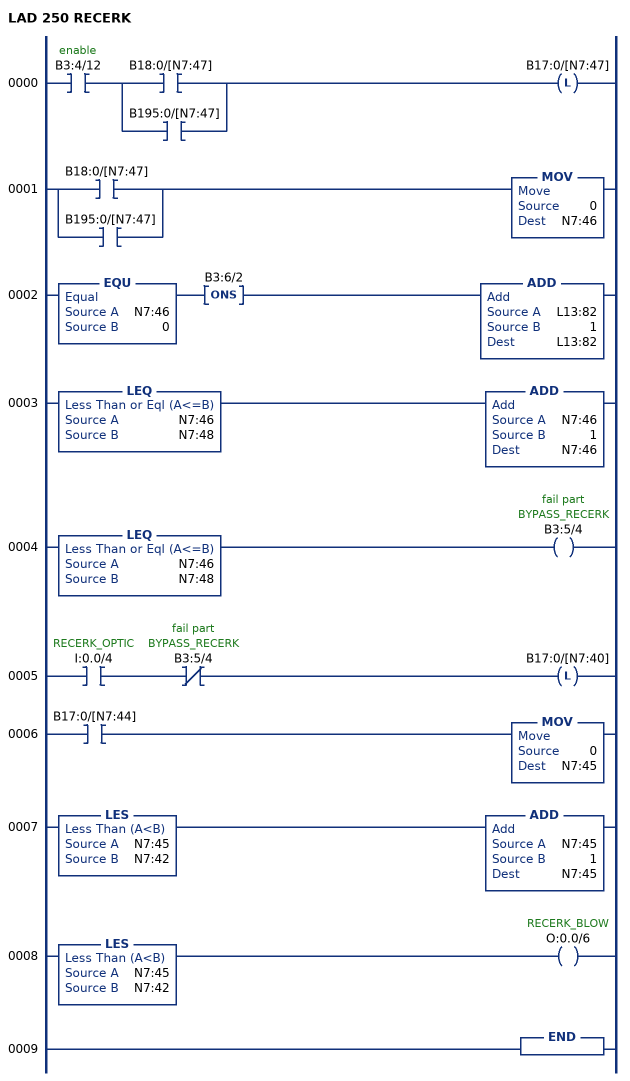
% Rung: 0 %
SOR XIC B3:4/12 BST XIC B18:0/[N7:47] NXB XIC B195:0/[N7:47] BND OTL B17:0/[N7:47] EOR
%   B3:4/12  "enable" %
%   B18:0  TOP_G %
%   N7:47  RECERK_BLOCKOPTIC_PT %
%   B195:0  TOP_NG %
%   B17:0  SIDE_G %
% Rung: 1 %
SOR BST XIC B18:0/[N7:47] NXB XIC B195:0/[N7:47] BND MOV 0 N7:46 EOR
%   B18:0  TOP_G %
%   N7:47  RECERK_BLOCKOPTIC_PT %
%   B195:0  TOP_NG %
% Rung: 2 %
SOR EQU N7:46 0 ONS B3:6/2 ADD L13:82 1 L13:82 EOR
% Rung: 3 %
SOR LEQ N7:46 N7:48 ADD N7:46 1 N7:46 EOR
%   N7:48  RECERK_BLK_BLOW_DIST %
% Rung: 4 %
SOR LEQ N7:46 N7:48 OTE B3:5/4 EOR
%   N7:48  RECERK_BLK_BLOW_DIST %
%   B3:5/4  BYPASS_RECERK  "fail part" %
% Rung: 5 %
SOR XIC I:0.0/4 XIO B3:5/4 OTL B17:0/[N7:40] EOR
%   I:0.0/4  RECERK_OPTIC %
%   B3:5/4  BYPASS_RECERK  "fail part" %
%   B17:0  SIDE_G %
%   N7:40  RECERK_OPTIC_POS %
% Rung: 6 %
SOR XIC B17:0/[N7:44] MOV 0 N7:45 EOR
%   B17:0  SIDE_G %
%   N7:44  RECERK_BLOW_POS  "adjusted for blow length" %
% Rung: 7 %
SOR LES N7:45 N7:42 ADD N7:45 1 N7:45 EOR
%   N7:42  RECERK_BLOW_LENGTH %
% Rung: 8 %
SOR LES N7:45 N7:42 OTE O:0.0/6 EOR
%   N7:42  RECERK_BLOW_LENGTH %
%   O:0.0/6  RECERK_BLOW %
% Rung: 9 %
SOR END EOR

LADDER 251 "RECERK SET"
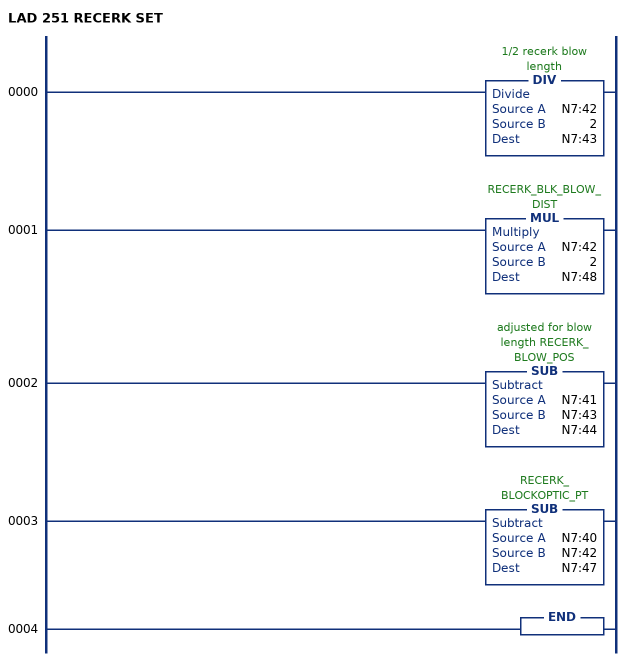
% Rung: 0 %
SOR DIV N7:42 2 N7:43 EOR
%   N7:42  RECERK_BLOW_LENGTH %
%   N7:43  "1/2 recerk blow length" %
% Rung: 1 %
SOR MUL N7:42 2 N7:48 EOR
%   N7:42  RECERK_BLOW_LENGTH %
%   N7:48  RECERK_BLK_BLOW_DIST %
% Rung: 2 %
SOR SUB N7:41 N7:43 N7:44 EOR
%   N7:41  RECERK_BLOW_POS_HMI  "recerk blow position set from hmi" %
%   N7:43  "1/2 recerk blow length" %
%   N7:44  RECERK_BLOW_POS  "adjusted for blow length" %
% Rung: 3 %
SOR SUB N7:40 N7:42 N7:47 EOR
%   N7:40  RECERK_OPTIC_POS %
%   N7:42  RECERK_BLOW_LENGTH %
%   N7:47  RECERK_BLOCKOPTIC_PT %
% Rung: 4 %
SOR END EOR

LADDER 252 "RATE1"
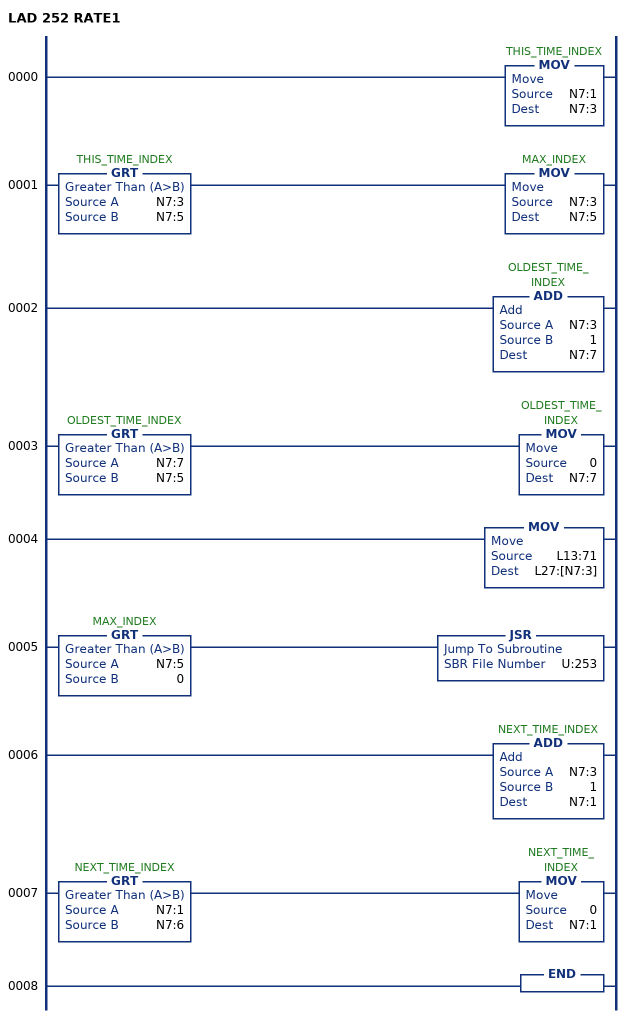
% Rung: 0 %
SOR MOV N7:1 N7:3 EOR
%   N7:1  NEXT_TIME_INDEX %
%   N7:3  THIS_TIME_INDEX %
% Rung: 1 %
SOR GRT N7:3 N7:5 MOV N7:3 N7:5 EOR
%   N7:3  THIS_TIME_INDEX %
%   N7:5  MAX_INDEX %
% Rung: 2 %
SOR ADD N7:3 1 N7:7 EOR
%   N7:3  THIS_TIME_INDEX %
%   N7:7  OLDEST_TIME_INDEX %
% Rung: 3 %
SOR GRT N7:7 N7:5 MOV 0 N7:7 EOR
%   N7:7  OLDEST_TIME_INDEX %
%   N7:5  MAX_INDEX %
% Rung: 4 %
SOR MOV L13:71 L27:[N7:3] EOR
%   L13:71  HSC_TIME %
%   N7:3  THIS_TIME_INDEX %
% Rung: 5 %
SOR GRT N7:5 0 JSR U:253 EOR
%   N7:5  MAX_INDEX %
% Rung: 6 %
SOR ADD N7:3 1 N7:1 EOR
%   N7:3  THIS_TIME_INDEX %
%   N7:1  NEXT_TIME_INDEX %
% Rung: 7 %
SOR GRT N7:1 N7:6 MOV 0 N7:1 EOR
%   N7:1  NEXT_TIME_INDEX %
%   N7:6  UPPER_INDEX_LIMIT  "buffer count 1" %
% Rung: 8 %
SOR END EOR

LADDER 253 "RATE2"
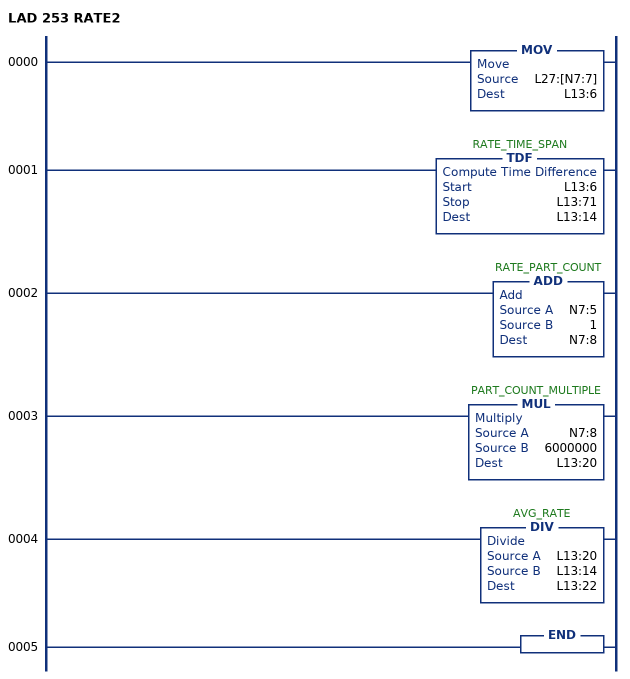
% Rung: 0 %
SOR MOV L27:[N7:7] L13:6 EOR
%   N7:7  OLDEST_TIME_INDEX %
% Rung: 1 %
SOR TDF L13:6 L13:71 L13:14 EOR
%   L13:71  HSC_TIME %
%   L13:14  RATE_TIME_SPAN %
% Rung: 2 %
SOR ADD N7:5 1 N7:8 EOR
%   N7:5  MAX_INDEX %
%   N7:8  RATE_PART_COUNT %
% Rung: 3 %
SOR MUL N7:8 6000000 L13:20 EOR
%   N7:8  RATE_PART_COUNT %
%   L13:20  PART_COUNT_MULTIPLE %
% Rung: 4 %
SOR DIV L13:20 L13:14 L13:22 EOR
%   L13:20  PART_COUNT_MULTIPLE %
%   L13:14  RATE_TIME_SPAN %
%   L13:22  AVG_RATE %
% Rung: 5 %
SOR END EOR

LADDER 254 "RESET RATE"
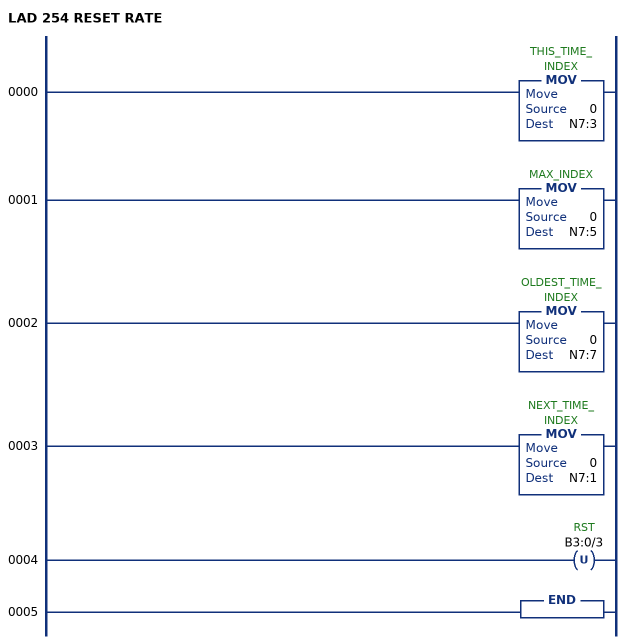
% Rung: 0 %
SOR MOV 0 N7:3 EOR
%   N7:3  THIS_TIME_INDEX %
% Rung: 1 %
SOR MOV 0 N7:5 EOR
%   N7:5  MAX_INDEX %
% Rung: 2 %
SOR MOV 0 N7:7 EOR
%   N7:7  OLDEST_TIME_INDEX %
% Rung: 3 %
SOR MOV 0 N7:1 EOR
%   N7:1  NEXT_TIME_INDEX %
% Rung: 4 %
SOR OTU B3:0/3 EOR
%   B3:0/3  RST %
% Rung: 5 %
SOR END EOR

LADDER 255 "UNUSED"
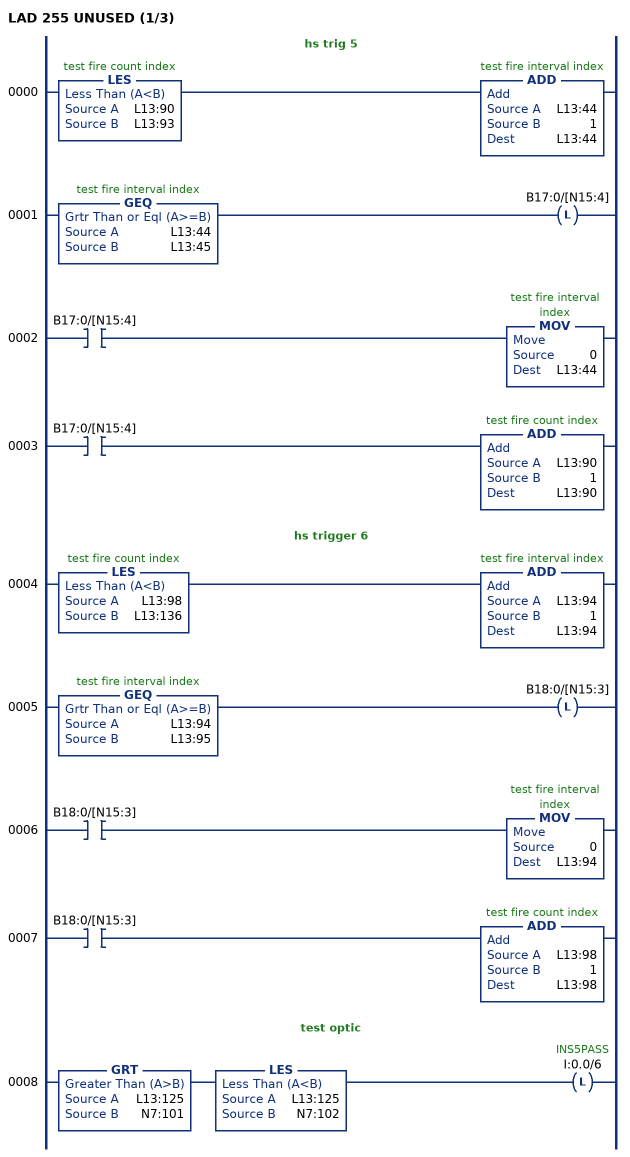
% Rung: 0 %
% TITLE: hs trig 5 %
SOR LES L13:90 L13:93 ADD L13:44 1 L13:44 EOR
%   L13:90  "test fire count index" %
%   L13:93  "test fire count" %
%   L13:44  "test fire interval index" %
% Rung: 1 %
SOR GEQ L13:44 L13:45 OTL B17:0/[N15:4] EOR
%   L13:44  "test fire interval index" %
%   L13:45  "test fire interval" %
%   B17:0  SIDE_G %
%   N15:4  INS_5_TRIG_LOC %
% Rung: 2 %
SOR XIC B17:0/[N15:4] MOV 0 L13:44 EOR
%   B17:0  SIDE_G %
%   N15:4  INS_5_TRIG_LOC %
%   L13:44  "test fire interval index" %
% Rung: 3 %
SOR XIC B17:0/[N15:4] ADD L13:90 1 L13:90 EOR
%   B17:0  SIDE_G %
%   N15:4  INS_5_TRIG_LOC %
%   L13:90  "test fire count index" %
% Rung: 4 %
% TITLE: hs trigger 6 %
SOR LES L13:98 L13:136 ADD L13:94 1 L13:94 EOR
%   L13:98  "test fire count index" %
%   L13:136  "test fire count" %
%   L13:94  "test fire interval index" %
% Rung: 5 %
SOR GEQ L13:94 L13:95 OTL B18:0/[N15:3] EOR
%   L13:94  "test fire interval index" %
%   L13:95  "test fire interval" %
%   B18:0  TOP_G %
%   N15:3  INS_6_TRIG_LOC %
% Rung: 6 %
SOR XIC B18:0/[N15:3] MOV 0 L13:94 EOR
%   B18:0  TOP_G %
%   N15:3  INS_6_TRIG_LOC %
%   L13:94  "test fire interval index" %
% Rung: 7 %
SOR XIC B18:0/[N15:3] ADD L13:98 1 L13:98 EOR
%   B18:0  TOP_G %
%   N15:3  INS_6_TRIG_LOC %
%   L13:98  "test fire count index" %
% Rung: 8 %
% TITLE: test optic %
SOR GRT L13:125 N7:101 LES L13:125 N7:102 OTL I:0.0/6 EOR
%   I:0.0/6  INS5PASS %

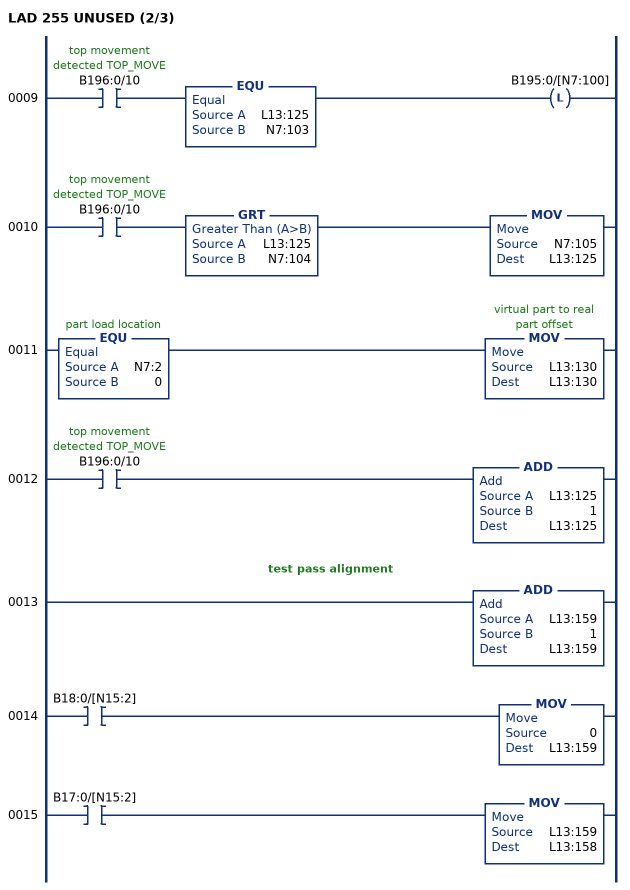
% Rung: 9 %
SOR XIC B196:0/10 EQU L13:125 N7:103 OTL B195:0/[N7:100] EOR
%   B196:0/10  TOP_MOVE  "top movement detected" %
%   B195:0  TOP_NG %
% Rung: 10 %
SOR XIC B196:0/10 GRT L13:125 N7:104 MOV N7:105 L13:125 EOR
%   B196:0/10  TOP_MOVE  "top movement detected" %
% Rung: 11 %
SOR EQU N7:2 0 MOV L13:130 L13:130 EOR
%   N7:2  "part load location" %
%   L13:130  "virtual part to real part offset" %
% Rung: 12 %
SOR XIC B196:0/10 ADD L13:125 1 L13:125 EOR
%   B196:0/10  TOP_MOVE  "top movement detected" %
% Rung: 13 %
% TITLE: test pass alignment %
SOR ADD L13:159 1 L13:159 EOR
% Rung: 14 %
SOR XIC B18:0/[N15:2] MOV 0 L13:159 EOR
%   B18:0  TOP_G %
%   N15:2  BLOW_PT %
% Rung: 15 %
SOR XIC B17:0/[N15:2] MOV L13:159 L13:158 EOR
%   B17:0  SIDE_G %
%   N15:2  BLOW_PT %

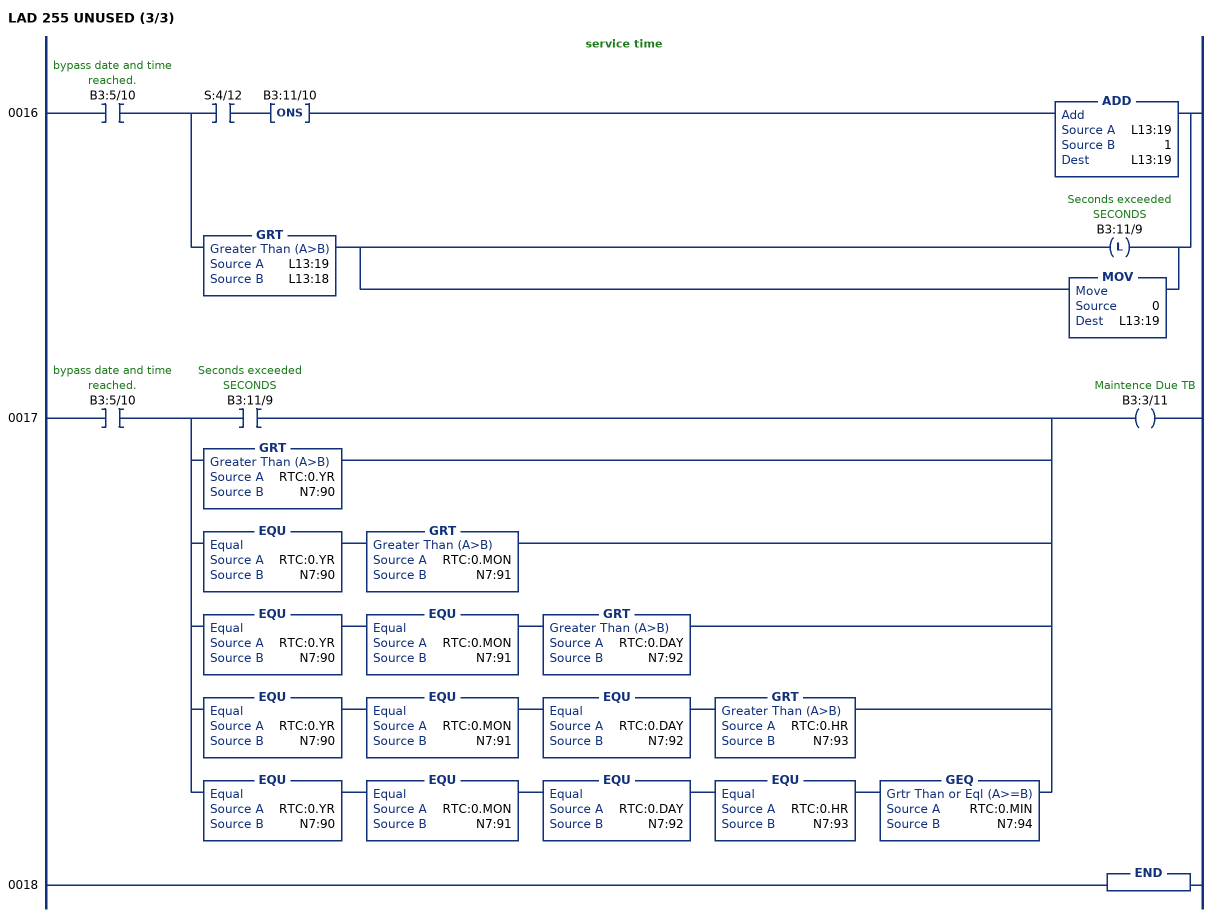
% Rung: 16 %
% TITLE: service time %
SOR XIC B3:5/10 BST XIC S:4/12 ONS B3:11/10 ADD L13:19 1 L13:19 NXB GRT L13:19 L13:18 BST OTL B3:11/9 NXB MOV 0 L13:19 BND BND EOR
%   B3:5/10  "bypass date and time reached." %
%   L13:18  MAX %
%   B3:11/9  SECONDS  "Seconds exceeded" %
% Rung: 17 %
SOR XIC B3:5/10 BST XIC B3:11/9 NXB GRT RTC:0.YR N7:90 NXB EQU RTC:0.YR N7:90 GRT RTC:0.MON N7:91 NXB EQU RTC:0.YR N7:90 EQU RTC:0.MON N7:91 GRT RTC:0.DAY N7:92 NXB EQU RTC:0.YR N7:90 EQU RTC:0.MON N7:91 EQU RTC:0.DAY N7:92 GRT RTC:0.HR N7:93 NXB EQU RTC:0.YR N7:90 EQU RTC:0.MON N7:91 EQU RTC:0.DAY N7:92 EQU RTC:0.HR N7:93 GEQ RTC:0.MIN N7:94 BND OTE B3:3/11 EOR
%   B3:5/10  "bypass date and time reached." %
%   B3:11/9  SECONDS  "Seconds exceeded" %
%   N7:90  RTC %
%   B3:3/11  TB  "Maintence Due" %
% Rung: 18 %
SOR END EOR

OTHER DOCUMENTED ADDRESSES
  B12:0/1  FELL_PARTS_FAULT
  B196:1/2  DOWNTRACK_OPTIC_RUN  "Feed Bowl optic Run Signal after timing delays"
  I:0.0/0  TOP_CONV_ENC_A
  I:0.0/1  TOP_CONV_ENC_B
  I:0.7  "Air Presure Sensor Input Signal"
  L13:61  "max acquisition time in ms"
  L42:0/2  "box full read (unused)"
  L42:1/1  "ps stop write (unused)"
  L183:3  L  "button state"
  N7:35  "maximum buffers"
  N15:9  FEED_WHEEL_STOP_TIME
  N197:7  "down track on delay"
  N197:8  "down track off delay"
  O:0.0/0  "spare"
  O:0.0/1  "spare"
  O:0.0/10  "spare"
  O:0.0/11  "spare"
  PFILE:6  "check for part jams"
  PFILE:10  "Bottom belt HSC"
  PFILE:12  "Top belt HSC"
  Q2:55  END_OF_MAIN
  T4:6  FEED_WHEEL_OFF_TIMER  "Delay to shut off feed wheel"
  U:6  "feed"
  U:217  "test trigger"

COMMENTS NOT ATTACHED TO A CURRENT RUNG
  F8:13: *************************
    Loads Side Camera Passing data into a bit shift
    *************************
    
    loads passing data bit into passing data bit shift register at the part present cl.
  I:0.0/8: special rung for testing. This rung can simulate a pass signal. It will not be timed correctly.
  B23:0/0: Yet another bit shift load with data in the part position indicating that there was a bottom system part pass as well as a top system part present at this location.
    
    verified works w/bypassed 071910 and unbypassed 072010
  C5:4: tempory counting to verify pass part count with boxing part count.
  B22:0/0: ***********************
     Bottom Part Syncronizing Logic
    ***********************
    
    This is the point at the bottom of the top conveyor where the part jumps from the bottom conveyor.  This system will then track the part through the top system to the point of the laser optic in order to verify that the part in question has passed the bottom inspection.  I believe that we NEED to include FAILING inspections to eliminate the possibility of a out of position part from passing. LW 072010
  T20:2.ACC: This rung is starting a timer that should be activated directly before the laser optic part presense sensor on the top conveyer and should cause the top optic to be ignored if the bottom camera system didn't pass. however other arrangements must be made if the bottom camera isn't going to be used as is the case with a nut inspection.
  T20:2: The timer used to verify that the part that triggered the top laser optic has passed the bottom camer. needs to be count
  N17:8: ****************************************************************************************************************
    I can not find anywhere in the program where the "Test Spacing From Pickup to Trigger is activated indicating to me that this entire function must not be doing anything in this program at this time.
    ****************************************************************************************************************
  B11:0/0: load part present bit shit with one shot data from the part present sensor
  B3:7/9: ************************************
     The next 3 rungs appear to do nothing
    ***********************************
  B3:6/1: ***********************
    Part Width and  Location
    ***********************
    
    Calculates the position of parts on the top belt by measureing the part width by calculating the number of belt movement pulses that occure when the optic is blocked and then devides that in half and add that to the optic location in the part presnet bit shift when the top optic is cleared.
  B9:0/[N7:47]: Remove any part present signals outside of expected location
  B9:0/[N7:50]: Remove any part present signals outside of expected location
  F19:0: Counter inside of a high speed counter interrupt counts the number of Bit Shifts that need to be processed in order to move the logic with the parts on the conveyor.
  F8:14: **************
    Bottom Top Camera Trigger
    *************
    
    Trigger Bottom Top Camera
  N10:4: test if boxing is connected
  B3:11/3: After initial delay allow blow two start functioning
  RUNG000150-000011: trigger count
  RUNG000150-000012: wipe stored part data if acq time expires
  RUNG000150-000013: clear data for aquire time expired
  RUNG000150-000014: clear data for time
  RUNG000150-000016: wiped count
  RUNG000150-000018: pass, fail and acquire inputs
  RUNG000150-000025: pass code / Set pass bit in Bit Shift
    captures result position and processing time
    Unlatch pass bit
  RUNG000150-000032: pass count
  RUNG000150-000035: fail count
  RUNG000150-000038: acquire code
  RUNG000150-000039: Grab trigger/acquire position
    Grab acquire time
  RUNG000150-000041: transfer tracked part positon from trigger/acquire to the acquire/result
    capture acquire time
    reset process time
  L14:8: on when ok for run
  L14:3: off when ok to run
  L14:2: off when ok to run
  L14:5: on when ok to run, rear off turns both off
  L13:165: maximum q i1
  N7:76: removed relieance on trigger signal
  N197:20/0: Passes deformed head blowoff command to TOP PLC where solenoid output is located.
  L13:162: maximum q
  L13:163: maximum average q
  B3:10/1: prevents momentary signals from box present sensor from tripping the logic for box not present
    
    This is in responce to a problem created by the sensor occasionally turning on as if no box was in its path when there is a box present.
  B3:6/2: IF PROCESSING FAULT OCURES AT COUNTER SENSOR; CLEAR THE BELT OF PASSING DATA
  L14:23: ****************  nEEDS fIXING  **********************
  L14:36: ****************  nEEDS fIXING  **********************
  RUNG000010-000014: ****
                      Zeros out the non passing part count when one passes
    ****
  RUNG000010-000018: Remove any part present signals outside of expected location
  T4:27: Check for buffer reset
  T4:26: Check for buffer reset
  RUNG000125-000014: clear data for time
  RUNG000125-000013: clear data for aquire time expired
  RUNG000125-000012: wipe stored part data if acq time expires
  RUNG000125-000011: trigger count
  RUNG000125-000029: Set pass bit in Bit Shift
    captures result position and processing time
    Unlatch pass bit
  RUNG000125-000027: transfer tracked part positon from trigger/acquire to the acquire/result
    capture acquire time
    reset process time
  RUNG000125-000026: Grab trigger/acquire position
    Grab acquire time
  RUNG000125-000025: pass code / Set pass bit in Bit Shift
    captures result position and processing time
    Unlatch pass bit
  RUNG000125-000018: pass, fail and acquire inputs
  RUNG000125-000016: wiped count

REVISION NOTES
  13: updated count reset
  14: added io moduals
  15: multiple steps toward new hmi integration
  21: test

DATA TABLE (non-zero values as saved)
DATA B3
% B3:0 % 0XA001 0X5060 0X02C4 0XA008 0X8B26 0X0341 0XA881 0X659A 0X4130 0X0000
% B3:10 % 0X2041 0X0846 0X2000 0X0000 0X0000 0X0000 0X0000 0X0000 0X0000 0X0000
DATA T4
% .PRE .ACC %
% T4:0 % 333 163
% T4:1 % 333 290
% T4:2 % 600 0
% T4:3 % 1000 1002
% T4:4 % 3 1
% T4:5 % 666 0
% T4:6 % 10 32766
% T4:7 % 250 0
% T4:8 % 250 0
% T4:9 % 50 3
% T4:10 % 200 0
% T4:11 % 666 0
% T4:12 % 14 29
% T4:13 % 6 4
% T4:14 % 250 0
% T4:15 % 333 30
% T4:16 % 333 19
% T4:17 % 100 64
% T4:18 % 120 120
% T4:19 % 300 0
% T4:20 % 200 0
% T4:21 % 200 0
% T4:22 % 200 0
% T4:23 % 250 0
% T4:24 % 666 0
% T4:25 % 666 0
% T4:26 % 250 0
% T4:27 % 250 0
% T4:28 % 250 0
% T4:29 % 5000 0
% T4:30 % 50 50
% T4:31 % 20 0
% T4:32 % 69 0
DATA C5
% .PRE .ACC %
% C5:0 % 32766 0
DATA R6
% .LEN .POS %
% R6:0 % 2048 0
% R6:1 % 2048 0
% R6:2 % 3 0
% R6:3 % 3 0
% R6:4 % 1250 0
% R6:5 % 1250 0
% R6:6 % 1300 0
% R6:7 % 10 0
% R6:8 % 3 0
% R6:9 % 3 0
% R6:10 % 1440 0
% R6:11 % 1440 0
% R6:12 % 10 0
% R6:13 % 10 0
% R6:14 % 10 0
% R6:15 % 10 0
% R6:16 % 1300 0
% R6:17 % 1440 0
% R6:18 % 1440 0
% R6:19 % 10 0
DATA N7
% N7:0 % 11069 27 1164 26 0 26 49 0 27 0
% N7:10 % 40 70 0 40 1512 250 777 666 10632 94
% N7:20 % 9591 93 9543 0 0 12 12 1580 333 20
% N7:30 % 46 10 2 20 46 10 1503 333 1493 333
% N7:40 % 2067 2122 40 20 2102 40 81 2027 80 1515
% N7:50 % 1520 400 27 14 0 0 32767 1520 28 15
% N7:60 % 1 1 4012 20 31 0 0 15 30 20
% N7:70 % 0 21 23 27738 32767 0 122 0 16 0
% N7:80 % 0 6 95 0 0 0 5 500 0 0
% N7:90 % 2011 4 4 12 1 0 0 0 0 1600
% N7:100 % 1003 90 110 100 175 25 0 0 0 0
DATA F8
% F8:0 % 18 206.64 23807 499 0.23807
% F8:5 % 0 0 500 1.9 2
% F8:10 % 1 0.08897486 0 101 63.26563
% F8:15 % 37.73437 4040 2 0 0
% F8:20 % 0 0.02 0 1 0
% F8:25 % 0 932781 0.222 279.6551 848597
% F8:30 % 0 170 0.03 38 852060
% F8:35 % 0 0 0 0 77
% F8:40 % 101 37.73437 0 100 1
% F8:45 % 1 2 0.21455 0 0
% F8:50 % 0 0 1 0 1
% F8:55 % 2000000 -221 0 0 0
% F8:95 % 0 0 0 492 4.92
DATA B12
% B12:0 % 0X0454 0X0000 0X0000 0X0000 0X0000 0X0000 0X0000 0X0000 0X0000 0X0000
DATA L13
% L13:0 % 308402300 308407124 4824 0 1000
% L13:5 % 1 -75983992 100 1162124017 1162124017
% L13:10 % 492 21600 28709 0 1030982652
% L13:15 % 350704886 -2147483648 2147483647 2147483647 82058
% L13:20 % 162000000 1592451203 0 320903532 1592451203
% L13:25 % 319 0 29801374 5 1000000000
% L13:30 % -344351 28623 1591069087 84 57344
% L13:35 % 0 57344 1591069087 1 1592451203
% L13:40 % -366691798 0 8 20 0
% L13:45 % 60 700 1 0 33
% L13:50 % 0 20 444 20 444
% L13:55 % 0 585 18048 10764 336
% L13:60 % 0 3300 84 2147483647 0
% L13:65 % 0 20 0 1926950760 1
% L13:70 % 955102215 955102183 32 0 2400
% L13:75 % -2 0 1072712 320903515 1073
% L13:80 % 319 -94 5615 0 2
% L13:85 % 6475 180 17292 344402 -463410
% L13:90 % 26616 0 0 1000 0
% L13:95 % 60 336 674 25989 350360221
% L13:100 % 351168041 -464527 -5036228 342295039 216
% L13:105 % 1592278120 1592278120 173083 0 537010368
% L13:110 % 6 1195 556 1590168231 1592376160
% L13:115 % 1592376187 27 14 1592376173 2207942
% L13:120 % 1195 3421 0 30 556
% L13:125 % 164 1592278120 1592278120 20 46
% L13:130 % 2207942 31204 31135 336 0
% L13:135 % 0 1000 337 12 0
% L13:140 % 12 6391320 12 0 20
% L13:145 % 64 1273 1284 111 111
% L13:150 % -1538760531 -1538760111 88 0 100
% L13:155 % 420 332 24 0 168160
% L13:160 % 3 18 4 395082 53203921
% L13:165 % 3 189116 95 13 8150
% L13:170 % 55946610 30 2868678 342419 0
% L13:175 % 0 0 45 32 38
% L13:180 % 176247033 25 99000 52866 644409
% L13:185 % 64 916459 92 627156 63
% L13:190 % 4 5 0 0 0
DATA F14
% F14:0 % 760.1599 200.1099 76 20 15
% F14:5 % 32766 21297.9 0 0 0
DATA N15
% N15:0 % 6 889 1976 1512 1502 134 100 1172 1150 10
% N15:10 % 61 504 0 0 0 0 1172 0 0 0
DATA L16
% L16:0 % 8 14 11 0 20
% L16:5 % 250 5000 5000 182 19
% L16:10 % 1256 18 2045 6599584 98
% L16:15 % 99 0 0 0 0
DATA B17
% B17:60 % 0XC000 0X0000 0X0000 0X0000 0X0000 0X0000 0X0000 0X0000 0X0000 0X0000
DATA B18
% B18:60 % 0XC000 0X0000 0X0000 0X0000 0X0000 0X0000 0X0000 0X0000 0X0000 0X0000
DATA L19
% L19:0 % -469940 -468592 -468256 -466907 -466571
% L19:5 % -465222 -464883 -381237 -380973 -380903
% L19:10 % -380854 -355115 -344351 -500587 -500251
% L19:15 % -498902 -498565 -497218 -496882 -495534
% L19:20 % -495198 -493853 -493515 -492169 -491833
% L19:25 % -490486 -490150 -488802 -488465 -487117
% L19:30 % -486780 -485430 -485093 -483747 -483408
% L19:35 % -482062 -481724 -480377 -480039 -478693
% L19:40 % -478357 -477010 -476673 -475325 -474988
% L19:45 % -473642 -473303 -471957 -471622 -470277
DATA L20
% L20:0 % 1592278120 1592278120 1592278120 1592278120 1592278120
% L20:5 % 1592278120 1592278120 1592294886 1592294950 1592294967
% L20:10 % 1592294979 1592301197 1592303799 1592278120 1592278120
% L20:15 % 1592278120 1592278120 1592278120 1592278120 1592278120
% L20:20 % 1592278120 1592278120 1592278120 1592278120 1592278120
% L20:25 % 1592278120 1592278120 1592278120 1592278120 1592278120
% L20:30 % 1592278120 1592278120 1592278120 1592278120 1592278120
% L20:35 % 1592278120 1592278120 1592278120 1592278120 1592278120
% L20:40 % 1592278120 1592278120 1592278120 1592278120 1592278120
% L20:45 % 1592278120 1592278120 1592278120 1592278120 1592278120
DATA L21
% L21:0 % 242620121 242621467 242621803 242623146 242623482
% L21:5 % 242624823 242625160 242626503 242626839 242628182
% L21:10 % 242628517 242629860 242630195 242631539 242631874
% L21:15 % 242633220 242633556 242634900 242635236 242636581
% L21:20 % 242636916 242638260 242638595 242822056 242822392
% L21:25 % 242822728 242823065 242823400 242823737 242824074
% L21:30 % 257003035 257003370 257003706 257005050 320901516
% L21:35 % 320901853 320902189 320902525 320902860 320903196
% L21:40 % 320903532 242613067 242613403 242614746 242615083
% L21:45 % 242616426 242616761 242618104 242618440 242619785
DATA L22
% L22:0 % 1592451203 1592451203 1592451203 1592451203 1592451203
% L22:5 % 1592451203 1592451203 1592451203 1592451203 1592451203
% L22:10 % 1592451203 1592451203 1592451203 1592451203 1592451203
% L22:15 % 1592451203 1592451203 1592451203 1592451203 1592451203
% L22:20 % 1592451203 1592451203 1592451203 1592451203 1592451203
% L22:25 % 1592451203 1592451203 1592451203 1592451203 1592451203
% L22:30 % 1592451203 1592451203 1592451203 1592451203 1592451203
% L22:35 % 1592451203 1592451203 1592451203 1592451203 1592451203
% L22:40 % 1592451203 1592451203 1592451203 1592451203 1592451203
% L22:45 % 1592451203 1592451203 1592451203 1592451203 1592451203
DATA L23
% L23:0 % 321208 322551 322887 324232 324567
% L23:5 % 325913 326249 327593 327929 329273
% L23:10 % 329610 330955 331291 332634 332970
% L23:15 % 334315 334651 335996 336332 337677
% L23:20 % 338014 339359 339694 341041 341377
% L23:25 % 342721 343058 344402 344738 304058
% L23:30 % 304394 305741 306077 307423 307759
% L23:35 % 309105 309442 310787 311123 312467
% L23:40 % 312803 314147 314482 315827 316163
% L23:45 % 317508 317844 319190 319527 320871
DATA L24
% L24:0 % 1592447007 1592447007 1592447007 1592447007 1592447007
% L24:5 % 1592447007 1592447007 1592447007 1592447007 1592447007
% L24:10 % 1592447007 1592447007 1592447007 1592447007 1592447007
% L24:15 % 1592447007 1592447007 1592447007 1592447007 1592447007
% L24:20 % 1592447007 1592447007 1592447007 1592447007 1592447007
% L24:25 % 1592447007 1592447007 1592447007 1592447007 1592447007
% L24:30 % 1592447007 1592447007 1592447007 1592447007 1592447007
% L24:35 % 1592447007 1592447007 1592447007 1592447007 1592447007
% L24:40 % 1592447007 1592447007 1592447007 1592447007 1592447007
% L24:45 % 1592447007 1592447007 1592447007 1592447007 1592447007
DATA L25
% L25:0 % -475206 -474868 -473520 -473183 -471837
% L25:5 % -471500 -470152 -469816 -468467 -468130
% L25:10 % -466782 -466444 -465096 -464759 -463410
% L25:15 % -463073 -503828 -503490 -502145 -501808
% L25:20 % -500462 -500127 -498781 -498444 -497099
% L25:25 % -496762 -495417 -495082 -493735 -493398
% L25:30 % -492050 -491712 -490368 -490032 -488687
% L25:35 % -488351 -487003 -486667 -485317 -484980
% L25:40 % -483630 -483292 -481947 -481608 -480262
% L25:45 % -479926 -478576 -478238 -476890 -476553
DATA L26
% L26:0 % 1592278120 1592278120 1592278120 1592278120 1592278120
% L26:5 % 1592278120 1592278120 1592278120 1592278120 1592278120
% L26:10 % 1592278120 1592278120 1592278120 1592278120 1592278120
% L26:15 % 1592278120 1592278120 1592278120 1592278120 1592278120
% L26:20 % 1592278120 1592278120 1592278120 1592278120 1592278120
% L26:25 % 1592278120 1592278120 1592278120 1592278120 1592278120
% L26:30 % 1592278120 1592278120 1592278120 1592278120 1592278120
% L26:35 % 1592278120 1592278120 1592278120 1592278120 1592278120
% L26:40 % 1592278120 1592278120 1592278120 1592278120 1592278120
% L26:45 % 1592278120 1592278120 1592278120 1592278120 1592278120
DATA L27
% L27:0 % -75983992 -75957196 -75956598 -75951544 -75950734
% L27:5 % -75947930 -75946415 -75945812 -75944870 -75943992
% L27:10 % -75941967 -75939459 -75934924 -75898731 -75897730
% L27:15 % -73346188 -72261338 -72201767 -68929091 -59219708
% L27:20 % -55819289 -53892544 -50990397 -48812047 -45021425
% L27:25 % -43383575 -41958136 502552452 531598359 531633864
% L27:30 % 531668449 531704205 531755229 531795341 531997256
% L27:35 % 625725685 625797461 627329145 627380790 627425916
% L27:40 % 627475622 627507784 627530557 627557972 627592344
% L27:45 % 627654448 627674800 627694163 627713711 627733603
DATA L42
% L42:0 % 8 256 0 0 0
% L42:5 % 45 45 45 0 0
% L42:20 % 0 0 32766 32766 0
% L42:50 % 0 30
DATA L183
% L183:0 % 1427522383 1427522384 1 1000000000 0
% L183:5 % 321 6 283 0 0
DATA N184
% N184:0 % 0 333 0 0 0 0 0 0 0 0
DATA B185
% B185:0 % 0X0200 0X0001 0X0000 0X0000 0X0000 0X0000 0X0000 0X0000 0X0000 0X0000
DATA N186
% N186:0 % 100 0 0 0 0 0 0 0 0 0
DATA L187
% L187:0 % 34 0 497 0 0
% L187:5 % 1063 0 0 0 0
DATA F188
% F188:0 % 6 66 11 44 29
DATA B189
% B189:0 % 0X00F0 0X0000 0X0000 0X0000 0X0000 0X0000 0X0000 0X0000 0X0000 0X0000
DATA L190
% L190:0 % 1 5 0 0 0
% L190:30 % 0 2 0 0 0
DATA B191
% B191:0 % 0X0000 0X0001 0X0000 0X0000 0X0000 0X0000 0X0000 0X0000 0X0000 0X0000
DATA L192
% L192:0 % -1444152502 266932201 5055 76 0
% L192:5 % 1000000 39200000 999 999 8
% L192:10 % 0 0 0 78 17
% L192:15 % 1926950760 332250347 860888 0 0
% L192:20 % 180 0 0 0 0
DATA F193
% F193:0 % 1.268652 0.315 0.022 6 760
% F193:5 % -0.8252563 0.2 -0.1650513 964.1756 31592.18
% F193:10 % 0.011 0.195 0.165 0.337 200
% F193:15 % 0.09407043 0.025 0.002351761 0 1092.66
DATA B196
% B196:0 % 0X0224 0X9FF2 0X0001 0X0000 0X0000 0X0000 0X0000 0X0000 0X0000 0X0000
% B196:30 % 0XE800 0X9BFF 0XEBFF 0XFFDF 0XFFFF 0X0000 0X0000 0X0000 0X0000 0X0000
DATA N197
% N197:0 % 1560 150 500 2500 2500 14417 5555 300 150 0
% N197:10 % 4000 969 4 0 0 0 0 0 0 0
% N197:30 % 15 48 0 0 0 0 0 0 0 0
DATA B198
% B198:0 % 0X0009 0X0000 0X0000 0X0000 0X0000 0X0000 0X0000 0X0000 0X0000 0X0000
DATA L199
% L199:0 % 1 5571998 134 11 3579521
% L199:5 % 0 0 0 5 43136
% L199:10 % 0 224 10256 556 0
% L199:15 % 0 0 0 278717848 518
% L199:20 % 28295 16430853 5001 5001 0
% L199:25 % 0 0 28329 1 3781224
% L199:30 % 21630086 251 3809367 15030467 111
% L199:35 % 555 555 0 0 0
DATA N200
% N200:0 % 2046 1231 985 2047 2045 1594 1241 2045 2045 2045
% N200:10 % 0 0 0 1277 178 2046 1000 2045 2045 1218
% N200:20 % 1555 0 0 0 0 0 0 0 0 0
% N200:30 % 0 0 32767 0 0 0 0 0 0 0
DATA L201
% L201:0 % 20 40 40 -3011735 44
% L201:5 % 96629277 0 0 -3010662 0
% L201:10 % 0 0 0 327 43
% L201:15 % 0 43 0 43 36830
DATA B202
% B202:0 % 0X2241 0X0000 0X0001 0X0000 0X0000 0X0000 0X0000 0X0000 0X0000 0X0000
DATA N203
% N203:0 % 115 115 116 333 334 333 444 0 445 444
% N203:10 % 555 556 555 0 0 0 0 0 0 0
DATA L204
% L204:0 % 333 333 333 1362 124
% L204:5 % 2000 2000 462 222 0
% L204:10 % 0 0 0 1327077052 1327077052
% L204:15 % 1327077052 1327077052 1 0 0
% L204:20 % 0 0 333 0 0
% L204:30 % 333 0 0 0 0
DATA F205
% F205:0 % 655.32 655.32 655.32 655.32 0
